Fanuc KAREL source: kt00959.KL

-- PROVISIONAL review KL for V1013-1; original PC SHA256 b7a74061e20f186f3a9c82d6e2132c7b91d46ab0e4cf98178297aaaf1faa3fd9
-- Incomplete behavior may be omitted. Consult companion uncertainty JSON. Do not deploy.
PROGRAM KT00959
%NOLOCKGROUP
VAR
  ENTRY : INTEGER
  PNAME : STRING[80]
  VNAME : STRING[80]
  STATUS : INTEGER
  VALUE : STRING[80]
BEGIN
  -- UNRESOLVED_PC offsets 5-12; opcodes 9C,23
  -- UNRESOLVED_PC offsets 17-25; opcodes 3F,75
  -- UNRESOLVED_PC offsets 30-43; opcodes 3F,75
  -- UNRESOLVED_PC offsets 48-88; opcodes 27,22,22,2A,22,2A,22,2A,22,B0
  -- UNRESOLVED_PC offsets 93-97; opcodes 7F
END KT00959
